ABB RobotStudio station: Smart Second  Behaviour.rspag

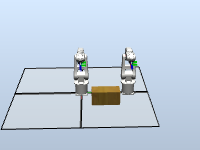
--- station ---
Station Multirobots - ABB 2 (saved by RobotStudio 6.8.8307.1040)
Controller Robot1
  mechanical unit ROB_1: IRB120_3_58__01, 6 joints, base frame (0, 0, 0) mm
Controller Robot2
  mechanical unit ROB_1: IRB120_3_58__01_2, 6 joints, base frame (0, 700, 0) mm
Layout (positions relative to the parent item):
  - IRB120_3_58__01 [mechanism, from Robots\IRB120_3_58_G_01.rslib] at (0, 0, 0) mm; joint values [0, -0.1323, 0.0406, 0, 0.6153, 0] (rad or m)
  - IRB120_3_58__01_2 [mechanism, from Robots\IRB120_3_58_G_01.rslib] at (0, 700, 0) mm; joint values [0, -0.1323, 0.0406, 0, 0.6153, 0] (rad or m)
  - Caja [part] at (0, 0, 0) mm
  - Componente inteligente_1 [smart component]
      signals: DI Detach, DI Attach
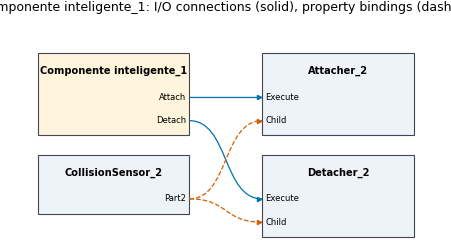
      connections:
        Componente inteligente_1.Attach -> Attacher_2.Execute
        Componente inteligente_1.Detach -> Detacher_2.Execute
        CollisionSensor_2.Part2 => Attacher_2.Child
        CollisionSensor_2.Part2 => Detacher_2.Child
    - Gripper [mechanism, from Libraries\Gripper.rslib] at (321.05, 0, 619) mm, rotated rx 180 ry 60 rz 180 deg
    - CollisionSensor_2 [smart component, from Components\CollisionSensor.rslib]
        properties: Object1=Gripper; Object2=(none); NearMiss=0.005; Part1=Gripper; Part2=Link5; CollisionType=2
    - Detacher_2 [smart component, from Components\Detacher.rslib]
        properties: Child=Link5; KeepPosition=true
    - Attacher_2 [smart component, from Components\Attacher.rslib]
        properties: Parent=Gripper; Flange=0; Child=Link5; Mount=false; Offset=[0 0 0]; Orientation=[0 0 0]
  - Componente inteligente_2 [smart component]
      signals: DI Attach, DI Detach
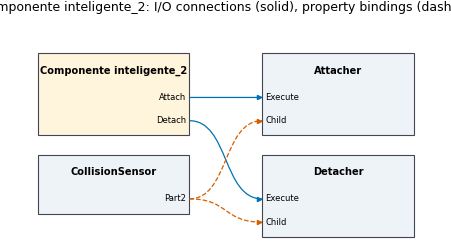
      connections:
        Componente inteligente_2.Attach -> Attacher.Execute
        Componente inteligente_2.Detach -> Detacher.Execute
        CollisionSensor.Part2 => Attacher.Child
        CollisionSensor.Part2 => Detacher.Child
    - Gripper2 [mechanism, from Libraries\Gripper2.rslib] at (321.05, 700, 619) mm, rotated rx 180 ry 60 rz 180 deg
    - CollisionSensor [smart component, from Components\CollisionSensor.rslib]
        properties: Object1=Gripper2; Object2=(none); NearMiss=0.005; Part1=Gripper2; Part2=Link6; CollisionType=2
    - Attacher [smart component, from Components\Attacher.rslib]
        properties: Parent=Gripper2; Flange=0; Child=Link6; Mount=false; Offset=[0 0 0]; Orientation=[0 0 0]
    - Detacher [smart component, from Components\Detacher.rslib]
        properties: Child=Link6; KeepPosition=true
Attachment: Gripper is attached to IRB120_3_58__01 / Link6
Attachment: Gripper2 is attached to IRB120_3_58__01_2 / Link6
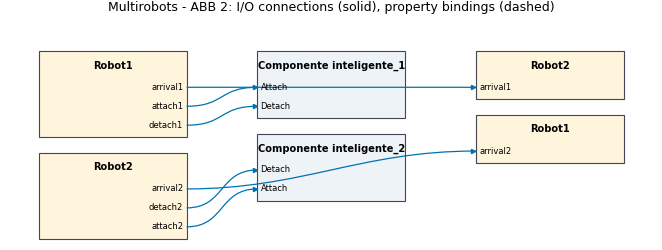
Station logic (signal -> signal, property => property):
  Robot1.arrival1 -> Robot2.arrival1
  Robot2.arrival2 -> Robot1.arrival2
  Robot1.attach1 -> Componente inteligente_1.Attach
  Robot1.detach1 -> Componente inteligente_1.Detach
  Robot2.detach2 -> Componente inteligente_2.Detach
  Robot2.attach2 -> Componente inteligente_2.Attach

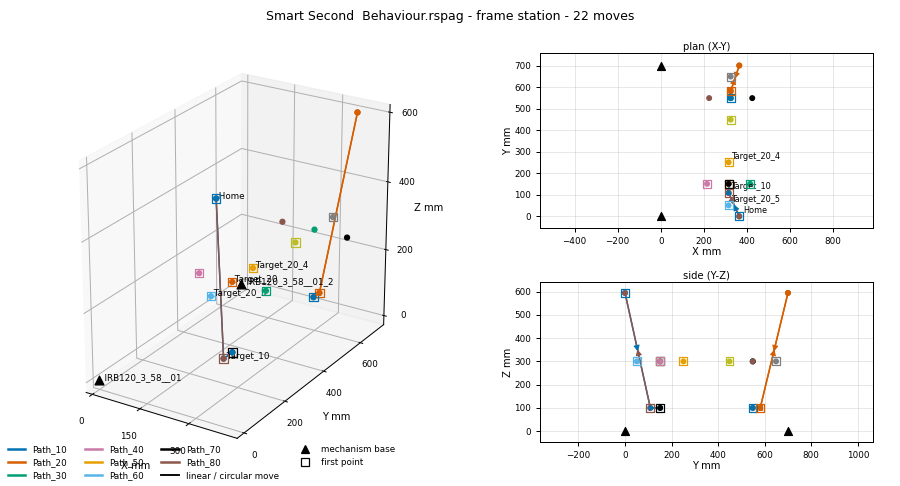
[picture p0: tool path of Smart Second  Behaviour.rspag in frame station, 22 of 22 moves have a stored position in this frame; points joined in program order, loops and branches not executed]
--- Backups/Robot1/RAPID/TASK1/PROGMOD/CalibData.mod ---
MODULE CalibData
	PERS tooldata Gripper:=[TRUE,[[0,0,50],[1,0,0,0]],[1,[0,0,1],[1,0,0,0],0,0,0]];
ENDMODULE

--- Backups/Robot1/RAPID/TASK1/PROGMOD/Module1.mod ---
MODULE Module1
	CONST robtarget Home:=[[364.353829072,0,594],[0.5,0,0.866025404,0],[0,0,0,0],[9E+09,9E+09,9E+09,9E+09,9E+09,9E+09]];
	CONST robtarget Target_10:=[[314.928,108.86,100],[0.707106781,-0.707106781,0,0],[0,0,0,0],[9E+09,9E+09,9E+09,9E+09,9E+09,9E+09]];
	CONST robtarget Target_10_2:=[[314.928,150.86,100],[0.707106781,-0.707106781,0,0],[0,0,0,0],[9E+09,9E+09,9E+09,9E+09,9E+09,9E+09]];
    CONST robtarget Target_20:=[[314.928,150.86,300],[0.707106781,-0.707106781,0,0],[0,0,0,0],[9E+09,9E+09,9E+09,9E+09,9E+09,9E+09]];
    CONST robtarget Target_20_2:=[[414.928,150.86,300],[0.707106781,-0.707106781,0,0],[0,0,0,0],[9E+09,9E+09,9E+09,9E+09,9E+09,9E+09]];
    CONST robtarget Target_20_3:=[[214.928,150.86,300],[0.707106781,-0.707106781,0,0],[0,0,0,0],[9E+09,9E+09,9E+09,9E+09,9E+09,9E+09]];
    CONST robtarget Target_20_4:=[[314.928,250.86,300],[0.707106781,-0.707106781,0,0],[0,0,0,0],[9E+09,9E+09,9E+09,9E+09,9E+09,9E+09]];
    CONST robtarget Target_20_5:=[[314.928,50.86,300],[0.707106781,-0.707106781,0,0],[0,0,0,0],[9E+09,9E+09,9E+09,9E+09,9E+09,9E+09]];
    !***********************************************************
    !
    ! Módulo:  Module1
    !
    ! Descripción:
    !   <Introduzca la descripción aquí>
    !
    ! Autor: Zuleika
    !
    ! Versión: 1.0
    !
    !***********************************************************


    !***********************************************************
    !
    ! Procedimiento Main
    !
    !   Este es el punto de entrada de su programa
    !
    !***********************************************************
    PROC main()
        SetDo arrival1, 0;

        Path_10;

        SetDo arrival1, 1;

        WaitDI arrival2, 1;
        SetDo arrival1, 0;

        PulseDO attach1;
        WaitTime 2;

        Path_20;

        SetDo arrival1, 1;

        WaitDI arrival2, 1;
        SetDo arrival1, 0;

        Path_30;

        SetDo arrival1, 1;

        WaitDI arrival2, 1;
        SetDo arrival1, 0;

        Path_40;

        SetDo arrival1, 1;

        WaitDI arrival2, 1;
        SetDo arrival1, 0;

        Path_50;

        SetDo arrival1, 1;

        WaitDI arrival2, 1;
        SetDo arrival1, 0;

        Path_60;

        SetDo arrival1, 1;

        WaitDI arrival2, 1;
        SetDo arrival1, 0;

        Path_70;

        SetDo arrival1, 1;

        WaitDI arrival2, 1;

        PulseDO detach1;
        WaitTime 2;

        Path_80;
    ENDPROC
	PROC Path_10()
	    MoveL Home,v300,z100,Gripper\WObj:=wobj0;
	    MoveL Target_10,v300,z0,Gripper\WObj:=wobj0;
	    MoveL Target_10_2,v150,fine,Gripper\WObj:=wobj0;
	ENDPROC
    PROC Path_20()
        MoveL Target_20,v150,fine,Gripper\WObj:=wobj0;
    ENDPROC
    PROC Path_30()
        MoveL Target_20_2,v150,fine,Gripper\WObj:=wobj0;
    ENDPROC
    PROC Path_40()
        MoveL Target_20_3,v150,fine,Gripper\WObj:=wobj0;
    ENDPROC
    PROC Path_50()
        MoveL Target_20_4,v150,fine,Gripper\WObj:=wobj0;
    ENDPROC
    PROC Path_60()
        MoveL Target_20_5,v150,fine,Gripper\WObj:=wobj0;
    ENDPROC
    PROC Path_70()
        MoveL Target_10_2,v150,fine,Gripper\WObj:=wobj0;
    ENDPROC
    PROC Path_80()
        MoveL Target_10,v300,z0,Gripper\WObj:=wobj0;
        MoveL Home,v300,z0,Gripper\WObj:=wobj0;
    ENDPROC
ENDMODULE

--- Backups/Robot2/RAPID/TASK1/PROGMOD/CalibData.mod ---
MODULE CalibData
	PERS tooldata Gripper2:=[TRUE,[[0,0,50],[1,0,0,0]],[1,[0,0,1],[1,0,0,0],0,0,0]];
ENDMODULE

--- Backups/Robot2/RAPID/TASK1/PROGMOD/Module1.mod ---
MODULE Module1
	CONST robtarget Home:=[[364.353829072,700,594],[0.5,0,0.866025404,0],[0,0,0,0],[9E+09,9E+09,9E+09,9E+09,9E+09,9E+09]];
	CONST robtarget Target_10:=[[324.584,580.767,100],[0.707106781,0.707106781,0,0],[-1,-2,-2,0],[9E+09,9E+09,9E+09,9E+09,9E+09,9E+09]];
	CONST robtarget Target_10_3:=[[324.584,550.767,100],[0.707106781,0.707106781,0,0],[-1,-2,-2,0],[9E+09,9E+09,9E+09,9E+09,9E+09,9E+09]];
    CONST robtarget Target_10_2:=[[324.584,548.767,100],[0.707106781,0.707106781,0,0],[-1,-2,-2,0],[9E+09,9E+09,9E+09,9E+09,9E+09,9E+09]];
    CONST robtarget Target_20:=[[324.584,548.767,300],[0.707106781,0.707106781,0,0],[-1,-2,-2,0],[9E+09,9E+09,9E+09,9E+09,9E+09,9E+09]];
    CONST robtarget Target_20_2:=[[424.584,548.767,300],[0.707106781,0.707106781,0,0],[-1,-2,-2,0],[9E+09,9E+09,9E+09,9E+09,9E+09,9E+09]];
    CONST robtarget Target_20_3:=[[224.584,548.767,300],[0.707106781,0.707106781,0,0],[-1,-2,-2,0],[9E+09,9E+09,9E+09,9E+09,9E+09,9E+09]];
    CONST robtarget Target_20_4:=[[324.584,648.767,300],[0.707106781,0.707106781,0,0],[-1,-2,-2,0],[9E+09,9E+09,9E+09,9E+09,9E+09,9E+09]];
    CONST robtarget Target_20_5:=[[324.584,448.767,300],[0.707106781,0.707106781,0,0],[-1,-2,-2,0],[9E+09,9E+09,9E+09,9E+09,9E+09,9E+09]];
    !***********************************************************
    !
    ! Módulo:  Module1
    !
    ! Descripción:
    !   <Introduzca la descripción aquí>
    !
    ! Autor: Zuleika
    !
    ! Versión: 1.0
    !
    !***********************************************************


    !***********************************************************
    !
    ! Procedimiento Main
    !
    !   Este es el punto de entrada de su programa
    !
    !***********************************************************
    PROC main()

        SetDO arrival2, 0;

        Path_20;

        SetDo arrival2, 1;

        WaitDI arrival1, 1;
        SetDO arrival2, 0;

        PulseDO attach2;
        WaitTime 2;

        Path_30;

        SetDo arrival2, 1;

        WaitDI arrival1, 1;
        SetDO arrival2, 0;

        Path_70;

        SetDo arrival2, 1;

        WaitDI arrival1, 1;
        SetDO arrival2, 0;

        Path_80;

        SetDo arrival2, 1;

        WaitDI arrival1, 1;
        SetDO arrival2, 0;

        Path_90;

        SetDo arrival2, 1;

        WaitDI arrival1, 1;
        SetDO arrival2, 0;

        Path_100;

        SetDo arrival2, 1;

        WaitDI arrival1, 1;
        SetDO arrival2, 0;

        Path_110;

        SetDo arrival2, 1;

        WaitDI arrival1, 1;

        PulseDO detach2;
        WaitTime 2;

        Path_120;

    ENDPROC
	PROC Path_20()
	    MoveL Home,v300,z100,Gripper2\WObj:=wobj0;
	    MoveL Target_10,v300,z0,Gripper2\WObj:=wobj0;
	    MoveL Target_10_2,v150,fine,Gripper2\WObj:=wobj0;
	ENDPROC
    PROC Path_30()
        MoveL Target_20,v150,fine,Gripper2\WObj:=wobj0;
    ENDPROC
    PROC Path_70()
        MoveL Target_20_2,v150,fine,Gripper2\WObj:=wobj0;
    ENDPROC
    PROC Path_80()
        MoveL Target_20_3,v150,fine,Gripper2\WObj:=wobj0;
    ENDPROC
    PROC Path_90()
        MoveL Target_20_4,v150,fine,Gripper2\WObj:=wobj0;
    ENDPROC
    PROC Path_100()
        MoveL Target_20_5,v150,fine,Gripper2\WObj:=wobj0;
    ENDPROC
    PROC Path_110()
        MoveL Target_10_2,v150,fine,Gripper2\WObj:=wobj0;
    ENDPROC
    PROC Path_120()
        MoveL Target_10,v300,z0,Gripper2\WObj:=wobj0;
        MoveL Home,v300,z0,Gripper2\WObj:=wobj0;
    ENDPROC
ENDMODULE

--- Backups/Robot1/SYSPAR/EIO.cfg ---
EIO:CFG_1.0:6:1::
#
EIO_SIGNAL:

      -Name "arrival1" -SignalType "DO"

      -Name "arrival2" -SignalType "DI"

      -Name "attach1" -SignalType "DO"

      -Name "detach1" -SignalType "DO"

--- Backups/Robot2/SYSPAR/EIO.cfg ---
EIO:CFG_1.0:6:1::
#
EIO_SIGNAL:

      -Name "arrival2" -SignalType "DO"

      -Name "arrival1" -SignalType "DI"

      -Name "attach2" -SignalType "DO"

      -Name "detach2" -SignalType "DO"
